FUNCTION location_PushBack : string
VAR_INPUT
	refdata : REFERENCE TO weather_data;
	refinput : REFERENCE TO STRING;
END_VAR
VAR
    nCommaPos : INT;
    nLen      : INT;
END_VAR

(* FUNC checks if provided string format is correct.*)
nCommaPos := FIND(refinput, ','); // returns 0 if not found
IF nCommaPos = 0 THEN
    RETURN;
END_IF

// Check length after comma
nLen := LEN(refinput);
IF (nLen - nCommaPos) = 2 THEN
	refdata.uLocIndex :=  refdata.uLocIndex + 1;
    refdata.sLocation[refdata.uLocIndex] := refinput;
END_IF

END_FUNCTION

(* stored: Version 1.1.0.1, ProductVersion 3.1.4024.15
   POU location_PushBack: Id {3dc8d68d-c871-4f2d-a1a8-bdd3872ba2d7}, SpecialFunc None *)
